Staubli VAL3: SMOVE.pgx

program SMOVE()
begin
  //
  while true
    if bruning==true and distart==true
      stopMove()
      bPause=true
      bruning=false
      wait(distart==false)
    endIf
    if bPause and distart==true
      restartMove()
      bruning=true
      bPause=false
      wait(distart==false)
    endIf
    delay(0)
  endWhile
end
